// TwinCAT 3 PLC project MAS418_PLC
// ProgramVersion: 3.1.4023.0
// libraries:
//   VisuSymbols,3.5.10.0,System
// project tree:
//   / GlobalTextList.TcGTLO, PlcTask.TcTTO, VisualizationManager.TcVMO (not stored)
//   POUs/ MAIN.TcPOU
//   VISUs/ HMI.TcVIS
// real-time tasks:
//   TASK PlcTask: cycle T#10ms, priority 20, ADS port 350

CONFIGURATION MAS418_PLC
    RESOURCE PLC ON TwinCAT3
        TASK PlcTask(INTERVAL := T#10ms, PRIORITY := 20);
        PROGRAM MAIN WITH PlcTask : MAIN;
    END_RESOURCE
END_CONFIGURATION

// ---- POUs/MAIN.TcPOU
PROGRAM MAIN
VAR
	bEnable : BOOL := FALSE;
	bStart : BOOL := FALSE; 
	switch: BOOL;
	Lamp: BOOL;
END_VAR

bEnable := bStart; 
bStart :=switch;
bEnable :=Lamp;

END_PROGRAM

// ---- VISUs/HMI.TcVIS
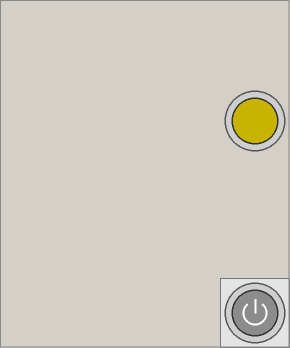
VISUALIZATION HMI  // 290x348
    Lamp1 (220,86 70x70), style: Lamp-Lamp1-Yellow
    PowerSwitch (220,278 70x70), behaviour: TOGGLE, style: Switch-PowerSwitch-Gray
END_VISUALIZATION
